# EPICS autosave request: iocBoot/sioc-li20-bl01/blen_manual.req
file "manual.req" AREA=LI20,POS=3014,INST=BZ203014A
file "manual.req" AREA=LI20,POS=3014,INST=BZ203014B
